(* Logix 5000 project; controller Sucrose_Main Emulate 5570 rev 20.12; software revision 20.01; part 20 of 30 *)
(* tags used below, declared in another part *)
   ClearFault_Master : BOOL;
   ClearFault_Master_TMR : TIMER;
   DATE_TIME : Date_Time;
   ONESHOTBITS : INT[10];
   Rung_Comment : BOOL;
   SucroseCIP_FILTRATION_REMOTE : CIP_REMOTE;
   SucroseDischarge : Area_Program;
   SucroseFiltration : Area_Program;
   TANK1_DATE_TIME : Date_Time;
   TANK2_DATE_TIME : Date_Time;
   TANK3_DATE_TIME : Date_Time;
   TK_23_01_01_RECEIVING_COMPLETE : BOOL;
   TK_23_02_01_RECEIVING_COMPLETE : BOOL;
   TK_23_03_01_RECEIVING_COMPLETE : BOOL;
(* Master_Main, continued *)

ROUTINE Date_Time   (* ladder *)
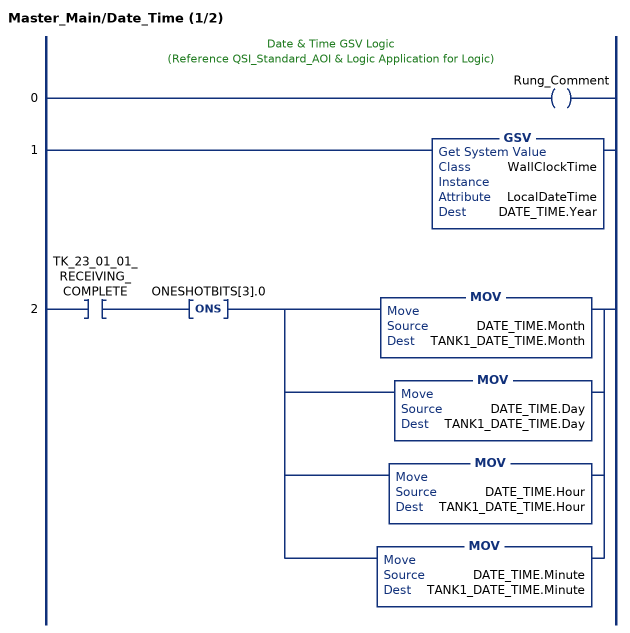
   // Date & Time GSV Logic
   // (Reference QSI_Standard_AOI & Logic Application for Logic)
   0: OTE(Rung_Comment);
   1: GSV(WallClockTime,,LocalDateTime,DATE_TIME.Year);
   2: XIC(TK_23_01_01_RECEIVING_COMPLETE)ONS(ONESHOTBITS[3].0)[MOV(DATE_TIME.Month,TANK1_DATE_TIME.Month) ,MOV(DATE_TIME.Day,TANK1_DATE_TIME.Day) ,MOV(DATE_TIME.Hour,TANK1_DATE_TIME.Hour) ,MOV(DATE_TIME.Minute,TANK1_DATE_TIME.Minute) ];
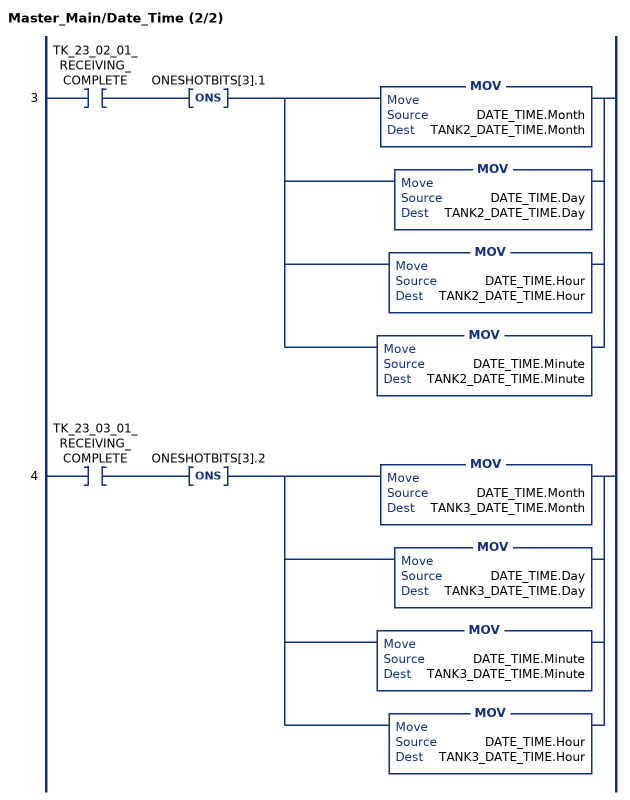
   3: XIC(TK_23_02_01_RECEIVING_COMPLETE)ONS(ONESHOTBITS[3].1)[MOV(DATE_TIME.Month,TANK2_DATE_TIME.Month) ,MOV(DATE_TIME.Day,TANK2_DATE_TIME.Day) ,MOV(DATE_TIME.Hour,TANK2_DATE_TIME.Hour) ,MOV(DATE_TIME.Minute,TANK2_DATE_TIME.Minute) ];
   4: XIC(TK_23_03_01_RECEIVING_COMPLETE)ONS(ONESHOTBITS[3].2)[MOV(DATE_TIME.Month,TANK3_DATE_TIME.Month) ,MOV(DATE_TIME.Day,TANK3_DATE_TIME.Day) ,MOV(DATE_TIME.Minute,TANK3_DATE_TIME.Minute) ,MOV(DATE_TIME.Hour,TANK3_DATE_TIME.Hour) ];
END_ROUTINE

ROUTINE Drive_ClearFault   (* ladder *)
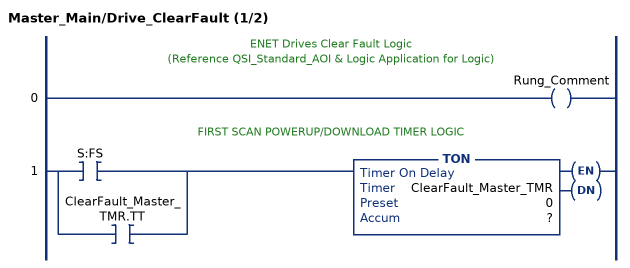
   // ENET Drives Clear Fault Logic
   // (Reference QSI_Standard_AOI & Logic Application for Logic)
   0: OTE(Rung_Comment);
   // FIRST SCAN POWERUP/DOWNLOAD TIMER LOGIC
   1: [XIC(S:FS) ,XIC(ClearFault_Master_TMR.TT) ]TON(ClearFault_Master_TMR,?,?);
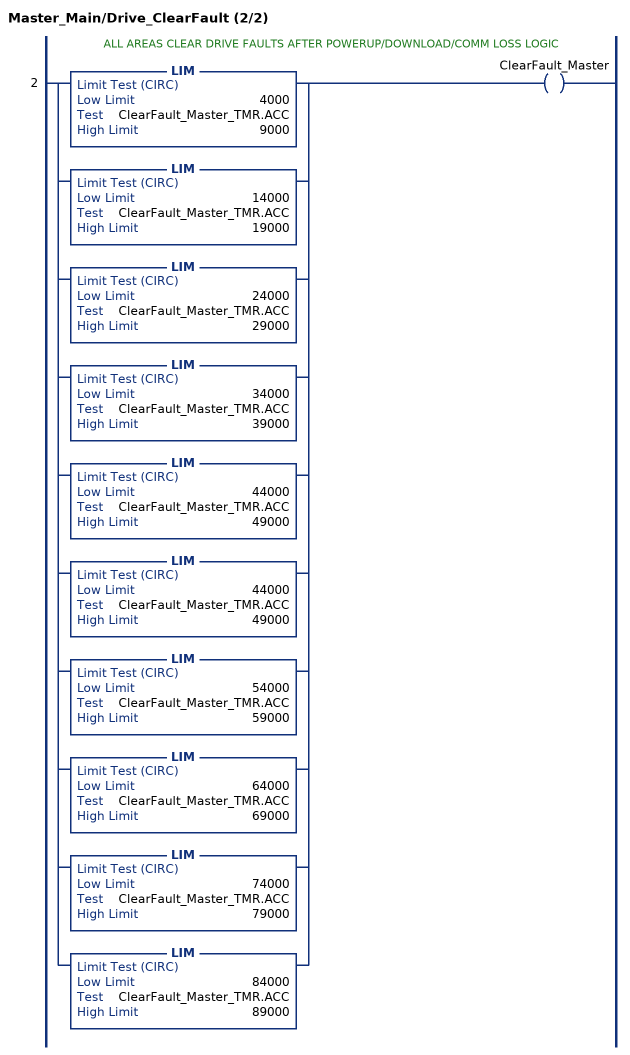
   // ALL AREAS CLEAR DRIVE FAULTS AFTER POWERUP/DOWNLOAD/COMM LOSS LOGIC
   2: [LIM(4000,ClearFault_Master_TMR.ACC,9000) ,LIM(14000,ClearFault_Master_TMR.ACC,19000) ,LIM(24000,ClearFault_Master_TMR.ACC,29000) ,LIM(34000,ClearFault_Master_TMR.ACC,39000) ,LIM(44000,ClearFault_Master_TMR.ACC,49000) ,LIM(44000,ClearFault_Master_TMR.ACC,49000) ,LIM(54000,ClearFault_Master_TMR.ACC,59000) ,LIM(64000,ClearFault_Master_TMR.ACC,69000) ,LIM(74000,ClearFault_Master_TMR.ACC,79000) ,LIM(84000,ClearFault_Master_TMR.ACC,89000) ]OTE(ClearFault_Master);
END_ROUTINE

ROUTINE HMI   (* ladder *)
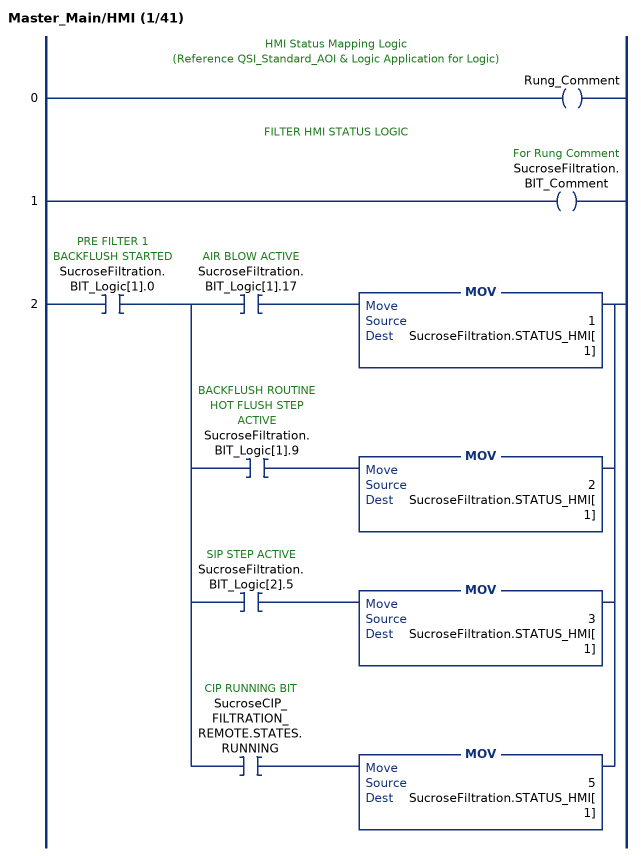
   // HMI Status Mapping Logic
   // (Reference QSI_Standard_AOI & Logic Application for Logic)
   0: OTE(Rung_Comment);
   // FILTER HMI STATUS LOGIC
   1: OTE(SucroseFiltration.BIT_Comment);
   2: XIC(SucroseFiltration.BIT_Logic[1].0)[XIC(SucroseFiltration.BIT_Logic[1].17) MOV(1,SucroseFiltration.STATUS_HMI[1]) ,XIC(SucroseFiltration.BIT_Logic[1].9) MOV(2,SucroseFiltration.STATUS_HMI[1]) ,XIC(SucroseFiltration.BIT_Logic[2].5) MOV(3,SucroseFiltration.STATUS_HMI[1]) ,XIC(SucroseCIP_FILTRATION_REMOTE.STATES.RUNNING) MOV(5,SucroseFiltration.STATUS_HMI[1]) ];
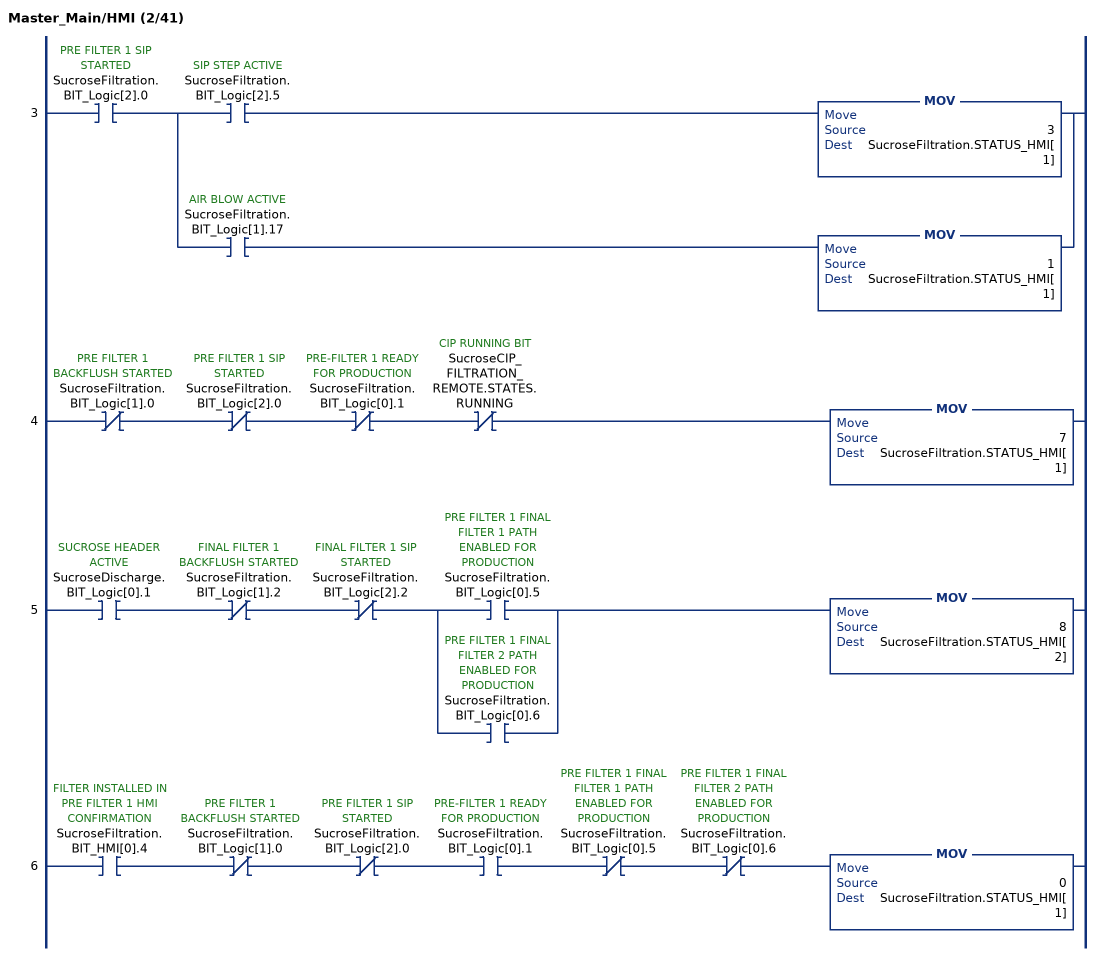
   3: XIC(SucroseFiltration.BIT_Logic[2].0)[XIC(SucroseFiltration.BIT_Logic[2].5) MOV(3,SucroseFiltration.STATUS_HMI[1]) ,XIC(SucroseFiltration.BIT_Logic[1].17) MOV(1,SucroseFiltration.STATUS_HMI[1]) ];
   4: XIO(SucroseFiltration.BIT_Logic[1].0)XIO(SucroseFiltration.BIT_Logic[2].0)XIO(SucroseFiltration.BIT_Logic[0].1)XIO(SucroseCIP_FILTRATION_REMOTE.STATES.RUNNING)MOV(7,SucroseFiltration.STATUS_HMI[1]);
   5: XIC(SucroseDischarge.BIT_Logic[0].1)XIO(SucroseFiltration.BIT_Logic[1].2)XIO(SucroseFiltration.BIT_Logic[2].2)[XIC(SucroseFiltration.BIT_Logic[0].5) ,XIC(SucroseFiltration.BIT_Logic[0].6) ]MOV(8,SucroseFiltration.STATUS_HMI[2]);
   6: XIC(SucroseFiltration.BIT_HMI[0].4)XIO(SucroseFiltration.BIT_Logic[1].0)XIO(SucroseFiltration.BIT_Logic[2].0)XIC(SucroseFiltration.BIT_Logic[0].1)XIO(SucroseFiltration.BIT_Logic[0].5)XIO(SucroseFiltration.BIT_Logic[0].6)MOV(0,SucroseFiltration.STATUS_HMI[1]);
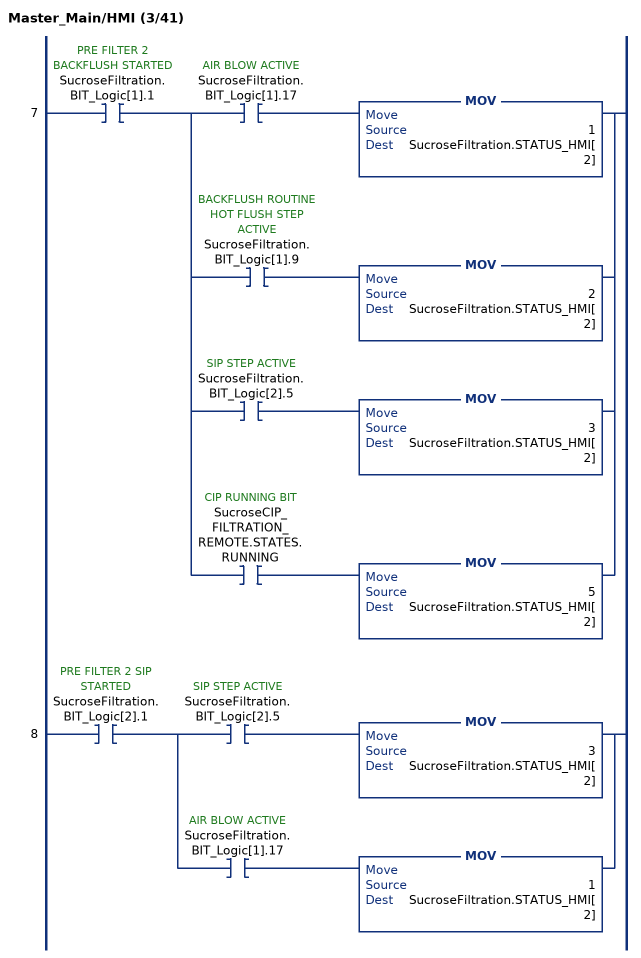
   7: XIC(SucroseFiltration.BIT_Logic[1].1)[XIC(SucroseFiltration.BIT_Logic[1].17) MOV(1,SucroseFiltration.STATUS_HMI[2]) ,XIC(SucroseFiltration.BIT_Logic[1].9) MOV(2,SucroseFiltration.STATUS_HMI[2]) ,XIC(SucroseFiltration.BIT_Logic[2].5) MOV(3,SucroseFiltration.STATUS_HMI[2]) ,XIC(SucroseCIP_FILTRATION_REMOTE.STATES.RUNNING) MOV(5,SucroseFiltration.STATUS_HMI[2]) ];
   8: XIC(SucroseFiltration.BIT_Logic[2].1)[XIC(SucroseFiltration.BIT_Logic[2].5) MOV(3,SucroseFiltration.STATUS_HMI[2]) ,XIC(SucroseFiltration.BIT_Logic[1].17) MOV(1,SucroseFiltration.STATUS_HMI[2]) ];
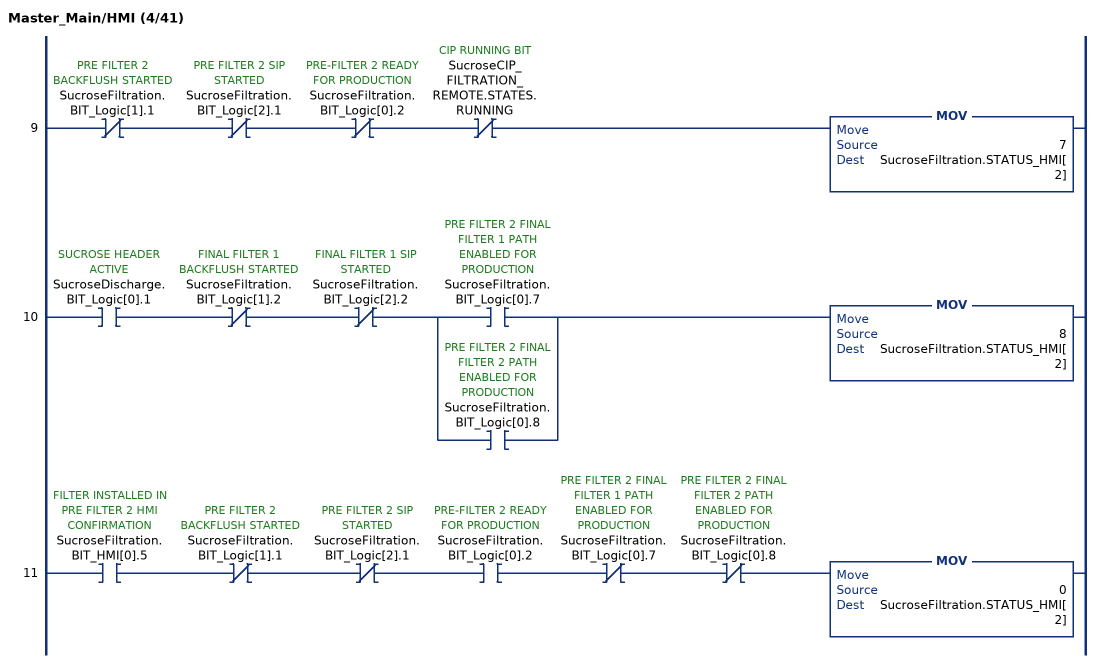
   9: XIO(SucroseFiltration.BIT_Logic[1].1)XIO(SucroseFiltration.BIT_Logic[2].1)XIO(SucroseFiltration.BIT_Logic[0].2)XIO(SucroseCIP_FILTRATION_REMOTE.STATES.RUNNING)MOV(7,SucroseFiltration.STATUS_HMI[2]);
   10: XIC(SucroseDischarge.BIT_Logic[0].1)XIO(SucroseFiltration.BIT_Logic[1].2)XIO(SucroseFiltration.BIT_Logic[2].2)[XIC(SucroseFiltration.BIT_Logic[0].7) ,XIC(SucroseFiltration.BIT_Logic[0].8) ]MOV(8,SucroseFiltration.STATUS_HMI[2]);
   11: XIC(SucroseFiltration.BIT_HMI[0].5)XIO(SucroseFiltration.BIT_Logic[1].1)XIO(SucroseFiltration.BIT_Logic[2].1)XIC(SucroseFiltration.BIT_Logic[0].2)XIO(SucroseFiltration.BIT_Logic[0].7)XIO(SucroseFiltration.BIT_Logic[0].8)MOV(0,SucroseFiltration.STATUS_HMI[2]);
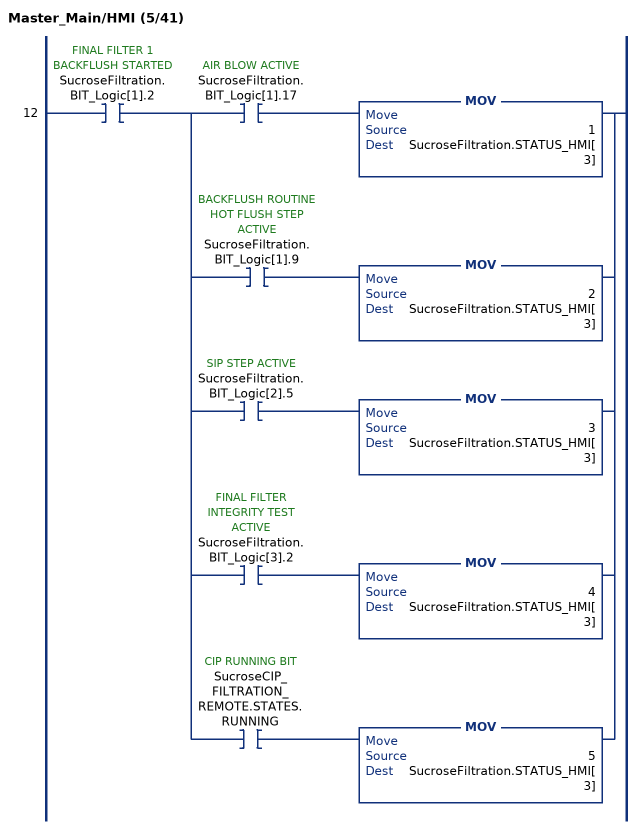
   12: XIC(SucroseFiltration.BIT_Logic[1].2)[XIC(SucroseFiltration.BIT_Logic[1].17) MOV(1,SucroseFiltration.STATUS_HMI[3]) ,XIC(SucroseFiltration.BIT_Logic[1].9) MOV(2,SucroseFiltration.STATUS_HMI[3]) ,XIC(SucroseFiltration.BIT_Logic[2].5) MOV(3,SucroseFiltration.STATUS_HMI[3]) ,XIC(SucroseFiltration.BIT_Logic[3].2) MOV(4,SucroseFiltration.STATUS_HMI[3]) ,XIC(SucroseCIP_FILTRATION_REMOTE.STATES.RUNNING) MOV(5,SucroseFiltration.STATUS_HMI[3]) ];
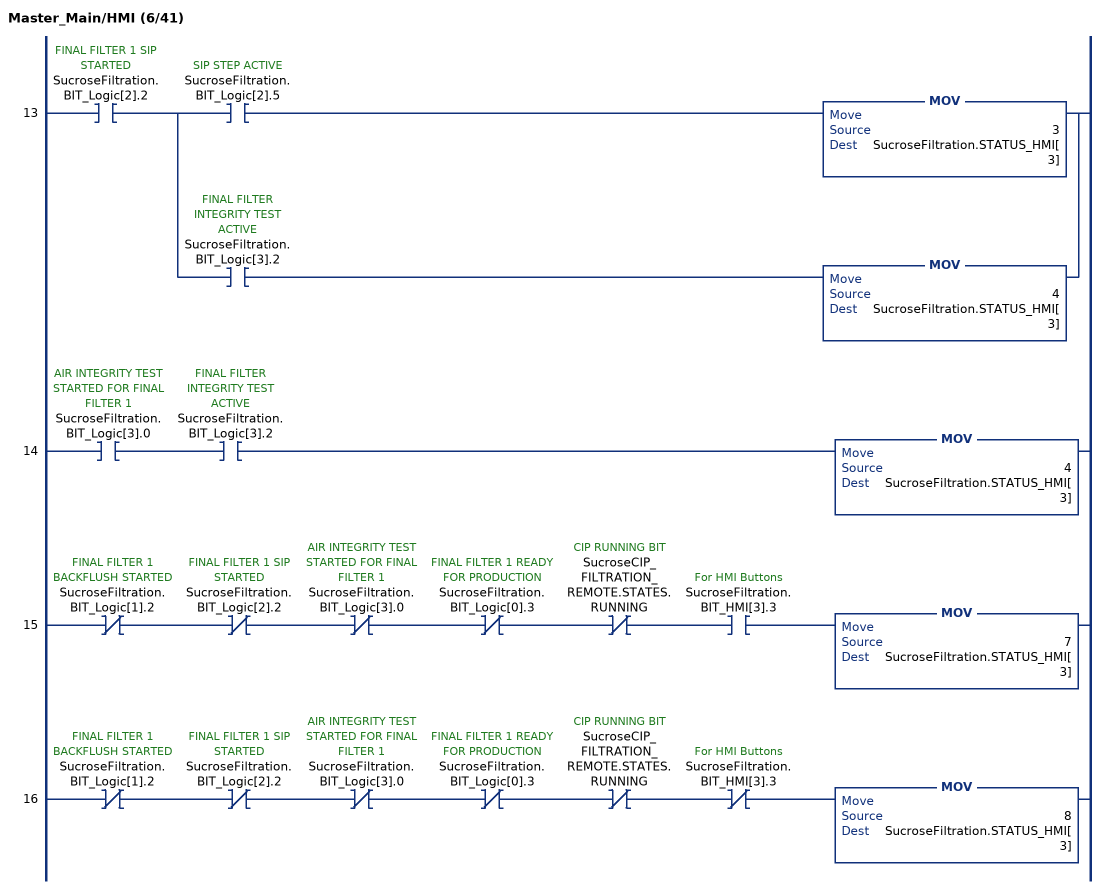
   13: XIC(SucroseFiltration.BIT_Logic[2].2)[XIC(SucroseFiltration.BIT_Logic[2].5) MOV(3,SucroseFiltration.STATUS_HMI[3]) ,XIC(SucroseFiltration.BIT_Logic[3].2) MOV(4,SucroseFiltration.STATUS_HMI[3]) ];
   14: XIC(SucroseFiltration.BIT_Logic[3].0)XIC(SucroseFiltration.BIT_Logic[3].2)MOV(4,SucroseFiltration.STATUS_HMI[3]);
   15: XIO(SucroseFiltration.BIT_Logic[1].2)XIO(SucroseFiltration.BIT_Logic[2].2)XIO(SucroseFiltration.BIT_Logic[3].0)XIO(SucroseFiltration.BIT_Logic[0].3)XIO(SucroseCIP_FILTRATION_REMOTE.STATES.RUNNING)XIC(SucroseFiltration.BIT_HMI[3].3)MOV(7,SucroseFiltration.STATUS_HMI[3]);
   16: XIO(SucroseFiltration.BIT_Logic[1].2)XIO(SucroseFiltration.BIT_Logic[2].2)XIO(SucroseFiltration.BIT_Logic[3].0)XIO(SucroseFiltration.BIT_Logic[0].3)XIO(SucroseCIP_FILTRATION_REMOTE.STATES.RUNNING)XIO(SucroseFiltration.BIT_HMI[3].3)MOV(8,SucroseFiltration.STATUS_HMI[3]);
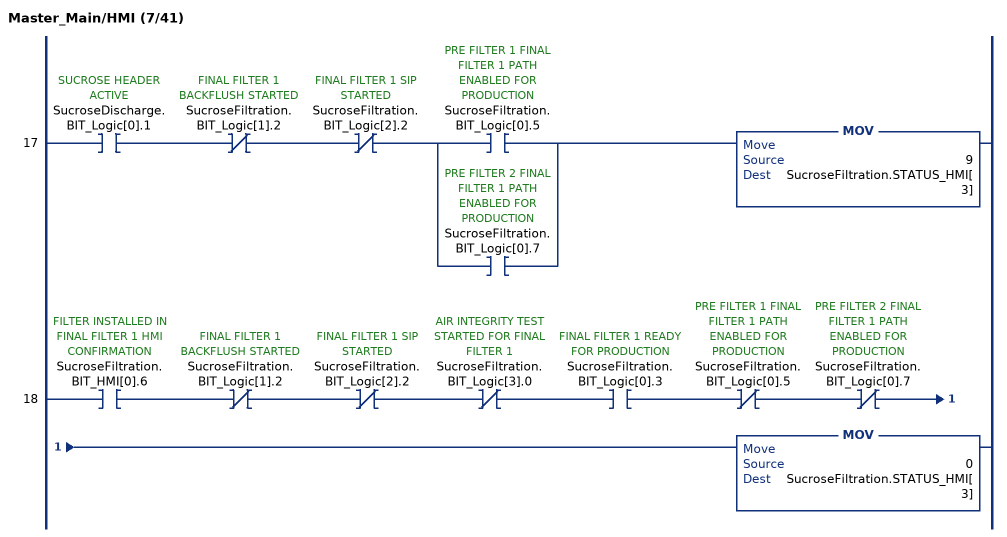
   17: XIC(SucroseDischarge.BIT_Logic[0].1)XIO(SucroseFiltration.BIT_Logic[1].2)XIO(SucroseFiltration.BIT_Logic[2].2)[XIC(SucroseFiltration.BIT_Logic[0].5) ,XIC(SucroseFiltration.BIT_Logic[0].7) ]MOV(9,SucroseFiltration.STATUS_HMI[3]);
   18: XIC(SucroseFiltration.BIT_HMI[0].6)XIO(SucroseFiltration.BIT_Logic[1].2)XIO(SucroseFiltration.BIT_Logic[2].2)XIO(SucroseFiltration.BIT_Logic[3].0)XIC(SucroseFiltration.BIT_Logic[0].3)XIO(SucroseFiltration.BIT_Logic[0].5)XIO(SucroseFiltration.BIT_Logic[0].7)MOV(0,SucroseFiltration.STATUS_HMI[3]);
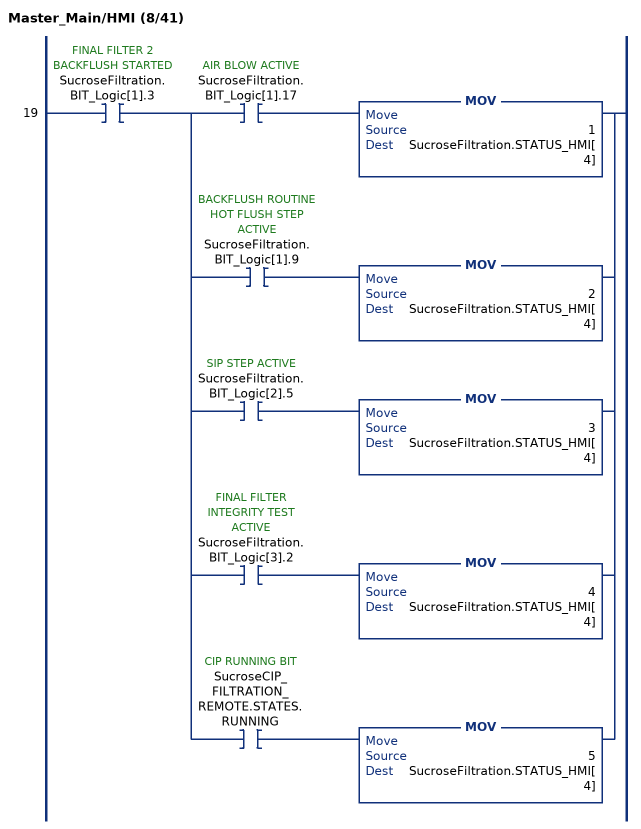
   19: XIC(SucroseFiltration.BIT_Logic[1].3)[XIC(SucroseFiltration.BIT_Logic[1].17) MOV(1,SucroseFiltration.STATUS_HMI[4]) ,XIC(SucroseFiltration.BIT_Logic[1].9) MOV(2,SucroseFiltration.STATUS_HMI[4]) ,XIC(SucroseFiltration.BIT_Logic[2].5) MOV(3,SucroseFiltration.STATUS_HMI[4]) ,XIC(SucroseFiltration.BIT_Logic[3].2) MOV(4,SucroseFiltration.STATUS_HMI[4]) ,XIC(SucroseCIP_FILTRATION_REMOTE.STATES.RUNNING) MOV(5,SucroseFiltration.STATUS_HMI[4]) ];
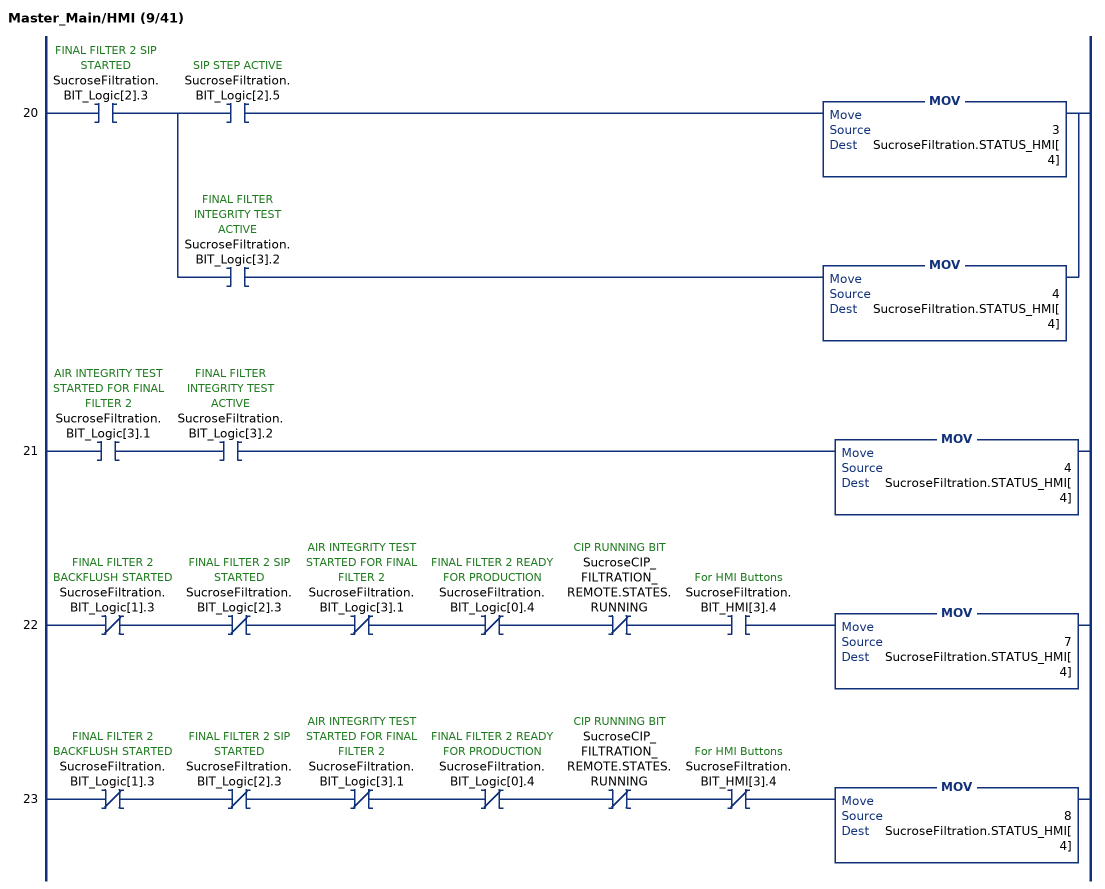
   20: XIC(SucroseFiltration.BIT_Logic[2].3)[XIC(SucroseFiltration.BIT_Logic[2].5) MOV(3,SucroseFiltration.STATUS_HMI[4]) ,XIC(SucroseFiltration.BIT_Logic[3].2) MOV(4,SucroseFiltration.STATUS_HMI[4]) ];
   21: XIC(SucroseFiltration.BIT_Logic[3].1)XIC(SucroseFiltration.BIT_Logic[3].2)MOV(4,SucroseFiltration.STATUS_HMI[4]);
   22: XIO(SucroseFiltration.BIT_Logic[1].3)XIO(SucroseFiltration.BIT_Logic[2].3)XIO(SucroseFiltration.BIT_Logic[3].1)XIO(SucroseFiltration.BIT_Logic[0].4)XIO(SucroseCIP_FILTRATION_REMOTE.STATES.RUNNING)XIC(SucroseFiltration.BIT_HMI[3].4)MOV(7,SucroseFiltration.STATUS_HMI[4]);
   23: XIO(SucroseFiltration.BIT_Logic[1].3)XIO(SucroseFiltration.BIT_Logic[2].3)XIO(SucroseFiltration.BIT_Logic[3].1)XIO(SucroseFiltration.BIT_Logic[0].4)XIO(SucroseCIP_FILTRATION_REMOTE.STATES.RUNNING)XIO(SucroseFiltration.BIT_HMI[3].4)MOV(8,SucroseFiltration.STATUS_HMI[4]);
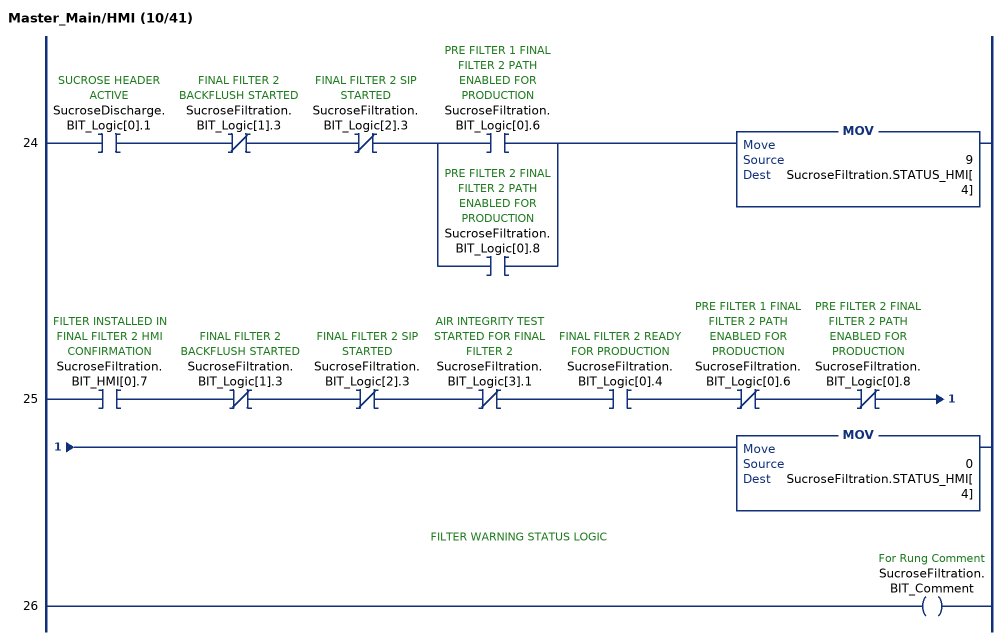
   24: XIC(SucroseDischarge.BIT_Logic[0].1)XIO(SucroseFiltration.BIT_Logic[1].3)XIO(SucroseFiltration.BIT_Logic[2].3)[XIC(SucroseFiltration.BIT_Logic[0].6) ,XIC(SucroseFiltration.BIT_Logic[0].8) ]MOV(9,SucroseFiltration.STATUS_HMI[4]);
   25: XIC(SucroseFiltration.BIT_HMI[0].7)XIO(SucroseFiltration.BIT_Logic[1].3)XIO(SucroseFiltration.BIT_Logic[2].3)XIO(SucroseFiltration.BIT_Logic[3].1)XIC(SucroseFiltration.BIT_Logic[0].4)XIO(SucroseFiltration.BIT_Logic[0].6)XIO(SucroseFiltration.BIT_Logic[0].8)MOV(0,SucroseFiltration.STATUS_HMI[4]);
   // FILTER WARNING STATUS LOGIC
   26: OTE(SucroseFiltration.BIT_Comment);
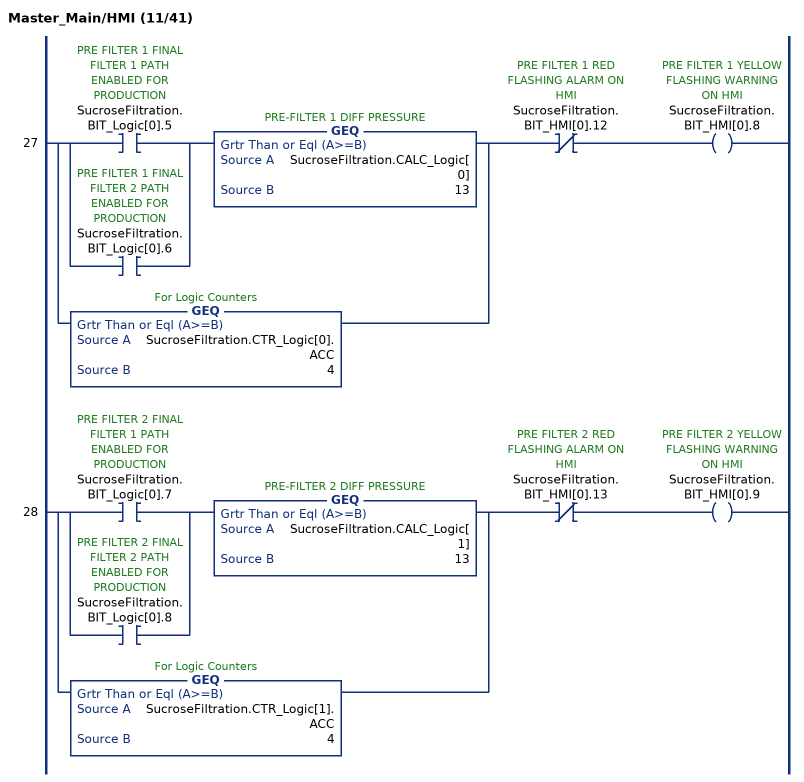
   27: [[XIC(SucroseFiltration.BIT_Logic[0].5) ,XIC(SucroseFiltration.BIT_Logic[0].6) ] GEQ(SucroseFiltration.CALC_Logic[0],13) ,GEQ(SucroseFiltration.CTR_Logic[0].ACC,4) ]XIO(SucroseFiltration.BIT_HMI[0].12)OTE(SucroseFiltration.BIT_HMI[0].8);
   28: [[XIC(SucroseFiltration.BIT_Logic[0].7) ,XIC(SucroseFiltration.BIT_Logic[0].8) ] GEQ(SucroseFiltration.CALC_Logic[1],13) ,GEQ(SucroseFiltration.CTR_Logic[1].ACC,4) ]XIO(SucroseFiltration.BIT_HMI[0].13)OTE(SucroseFiltration.BIT_HMI[0].9);
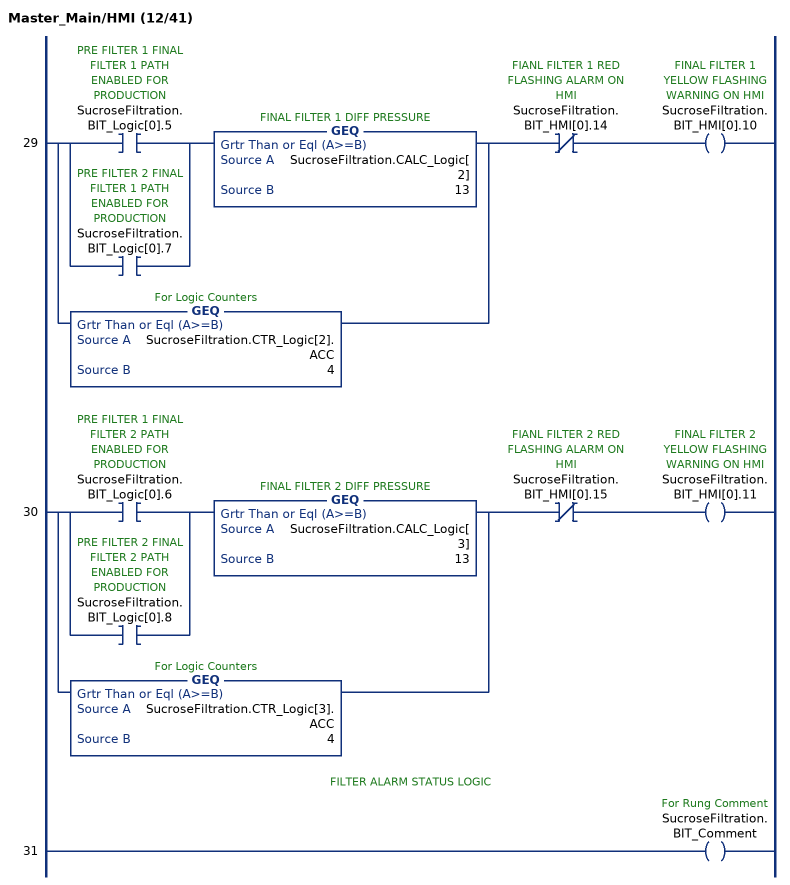
   29: [[XIC(SucroseFiltration.BIT_Logic[0].5) ,XIC(SucroseFiltration.BIT_Logic[0].7) ] GEQ(SucroseFiltration.CALC_Logic[2],13) ,GEQ(SucroseFiltration.CTR_Logic[2].ACC,4) ]XIO(SucroseFiltration.BIT_HMI[0].14)OTE(SucroseFiltration.BIT_HMI[0].10);
   30: [[XIC(SucroseFiltration.BIT_Logic[0].6) ,XIC(SucroseFiltration.BIT_Logic[0].8) ] GEQ(SucroseFiltration.CALC_Logic[3],13) ,GEQ(SucroseFiltration.CTR_Logic[3].ACC,4) ]XIO(SucroseFiltration.BIT_HMI[0].15)OTE(SucroseFiltration.BIT_HMI[0].11);
   // FILTER ALARM STATUS LOGIC
   31: OTE(SucroseFiltration.BIT_Comment);
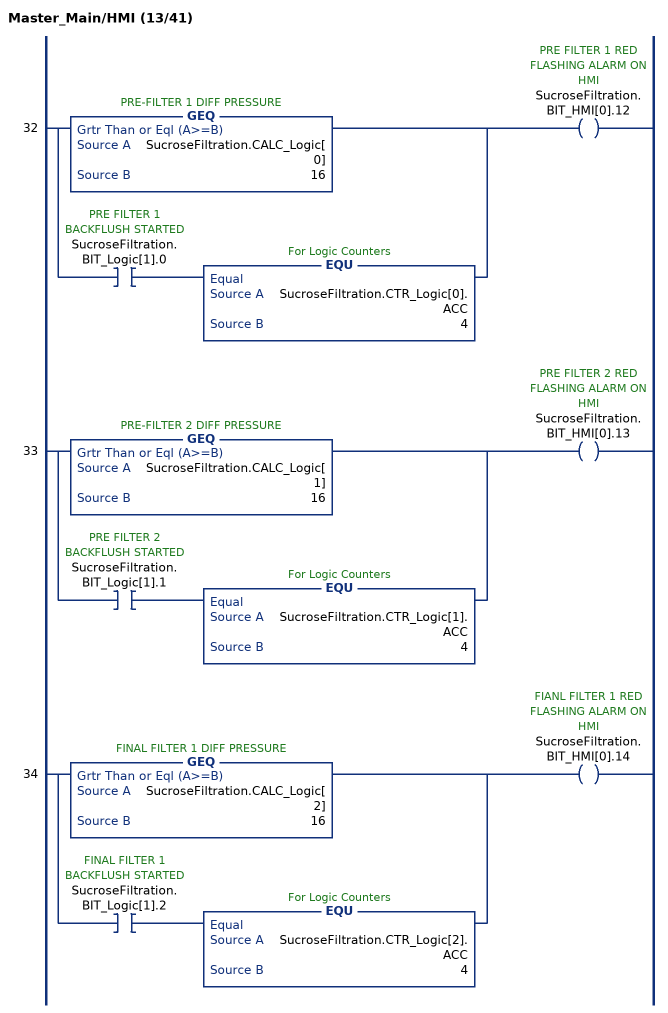
   32: [GEQ(SucroseFiltration.CALC_Logic[0],16) ,XIC(SucroseFiltration.BIT_Logic[1].0) EQU(SucroseFiltration.CTR_Logic[0].ACC,4) ]OTE(SucroseFiltration.BIT_HMI[0].12);
   33: [GEQ(SucroseFiltration.CALC_Logic[1],16) ,XIC(SucroseFiltration.BIT_Logic[1].1) EQU(SucroseFiltration.CTR_Logic[1].ACC,4) ]OTE(SucroseFiltration.BIT_HMI[0].13);
   34: [GEQ(SucroseFiltration.CALC_Logic[2],16) ,XIC(SucroseFiltration.BIT_Logic[1].2) EQU(SucroseFiltration.CTR_Logic[2].ACC,4) ]OTE(SucroseFiltration.BIT_HMI[0].14);
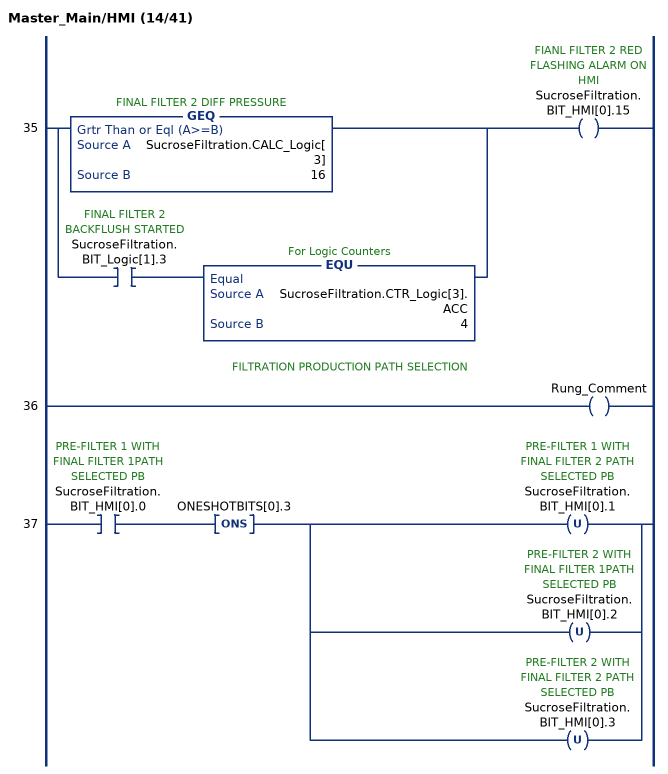
   35: [GEQ(SucroseFiltration.CALC_Logic[3],16) ,XIC(SucroseFiltration.BIT_Logic[1].3) EQU(SucroseFiltration.CTR_Logic[3].ACC,4) ]OTE(SucroseFiltration.BIT_HMI[0].15);
   // FILTRATION PRODUCTION PATH SELECTION
   36: OTE(Rung_Comment);
   37: XIC(SucroseFiltration.BIT_HMI[0].0)ONS(ONESHOTBITS[0].3)[OTU(SucroseFiltration.BIT_HMI[0].1) ,OTU(SucroseFiltration.BIT_HMI[0].2) ,OTU(SucroseFiltration.BIT_HMI[0].3) ];
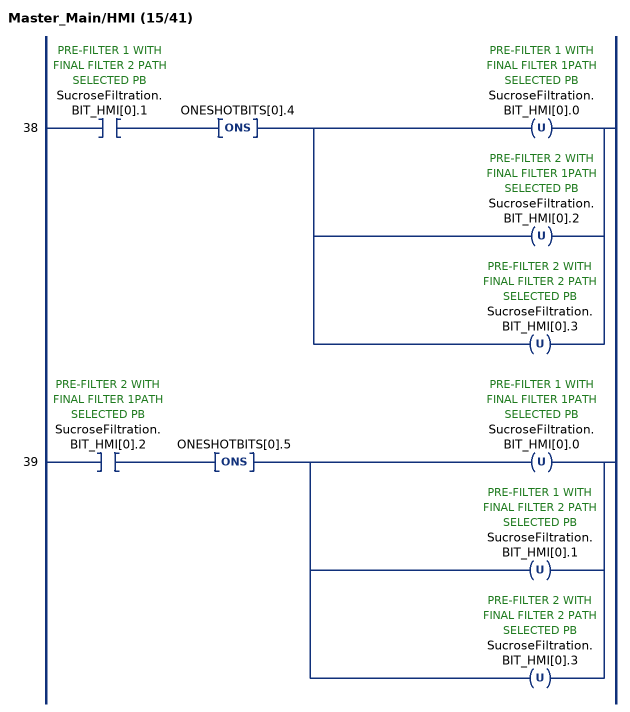
   38: XIC(SucroseFiltration.BIT_HMI[0].1)ONS(ONESHOTBITS[0].4)[OTU(SucroseFiltration.BIT_HMI[0].0) ,OTU(SucroseFiltration.BIT_HMI[0].2) ,OTU(SucroseFiltration.BIT_HMI[0].3) ];
   39: XIC(SucroseFiltration.BIT_HMI[0].2)ONS(ONESHOTBITS[0].5)[OTU(SucroseFiltration.BIT_HMI[0].0) ,OTU(SucroseFiltration.BIT_HMI[0].1) ,OTU(SucroseFiltration.BIT_HMI[0].3) ];
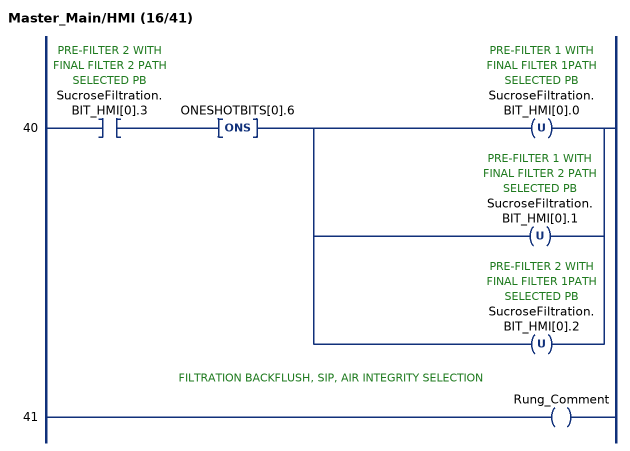
   40: XIC(SucroseFiltration.BIT_HMI[0].3)ONS(ONESHOTBITS[0].6)[OTU(SucroseFiltration.BIT_HMI[0].0) ,OTU(SucroseFiltration.BIT_HMI[0].1) ,OTU(SucroseFiltration.BIT_HMI[0].2) ];
   // FILTRATION BACKFLUSH, SIP, AIR INTEGRITY SELECTION
   41: OTE(Rung_Comment);
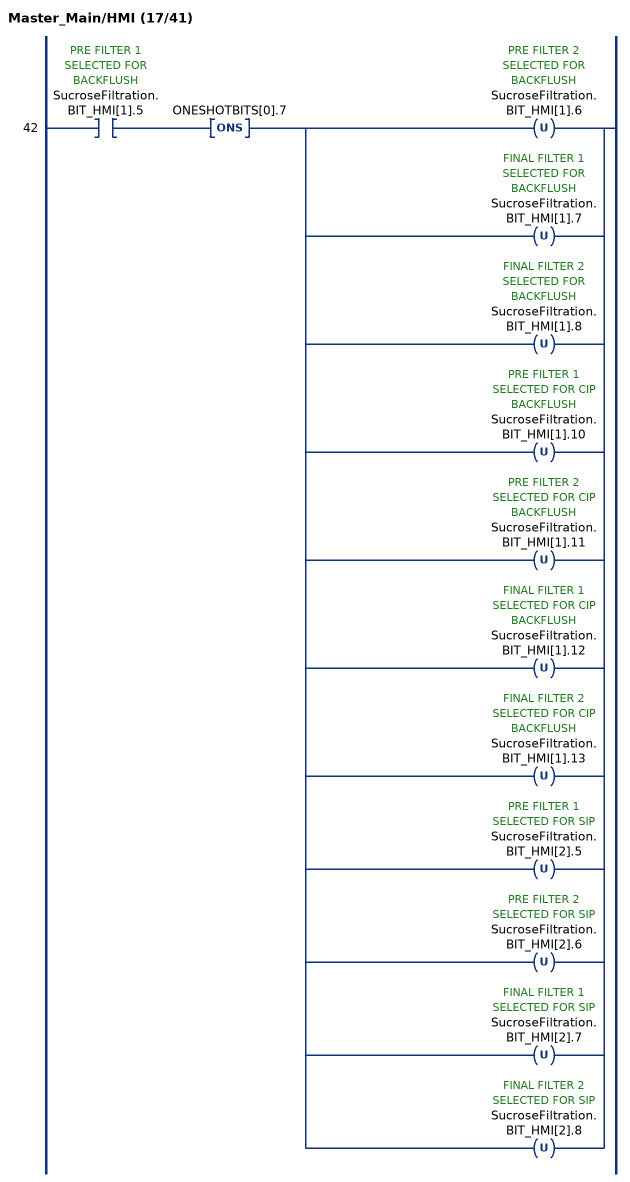
   42: XIC(SucroseFiltration.BIT_HMI[1].5)ONS(ONESHOTBITS[0].7)[OTU(SucroseFiltration.BIT_HMI[1].6) ,OTU(SucroseFiltration.BIT_HMI[1].7) ,OTU(SucroseFiltration.BIT_HMI[1].8) ,OTU(SucroseFiltration.BIT_HMI[1].10) ,OTU(SucroseFiltration.BIT_HMI[1].11) ,OTU(SucroseFiltration.BIT_HMI[1].12) ,OTU(SucroseFiltration.BIT_HMI[1].13) ,OTU(SucroseFiltration.BIT_HMI[2].5) ,OTU(SucroseFiltration.BIT_HMI[2].6) ,OTU(SucroseFiltration.BIT_HMI[2].7) ,OTU(SucroseFiltration.BIT_HMI[2].8) ];
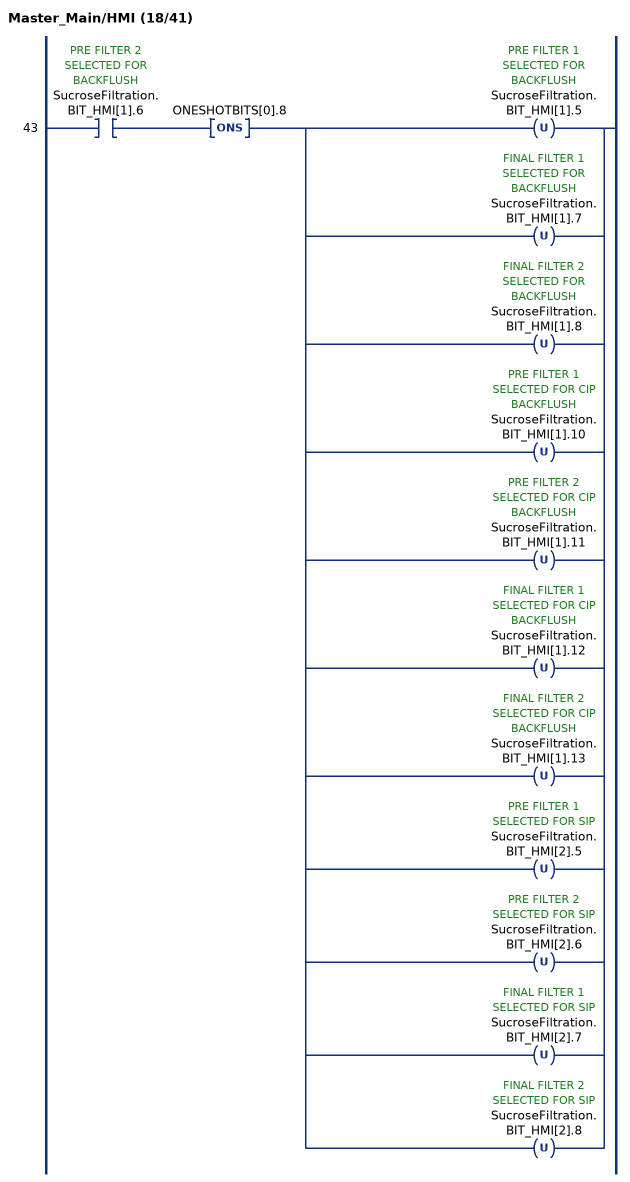
   43: XIC(SucroseFiltration.BIT_HMI[1].6)ONS(ONESHOTBITS[0].8)[OTU(SucroseFiltration.BIT_HMI[1].5) ,OTU(SucroseFiltration.BIT_HMI[1].7) ,OTU(SucroseFiltration.BIT_HMI[1].8) ,OTU(SucroseFiltration.BIT_HMI[1].10) ,OTU(SucroseFiltration.BIT_HMI[1].11) ,OTU(SucroseFiltration.BIT_HMI[1].12) ,OTU(SucroseFiltration.BIT_HMI[1].13) ,OTU(SucroseFiltration.BIT_HMI[2].5) ,OTU(SucroseFiltration.BIT_HMI[2].6) ,OTU(SucroseFiltration.BIT_HMI[2].7) ,OTU(SucroseFiltration.BIT_HMI[2].8) ];
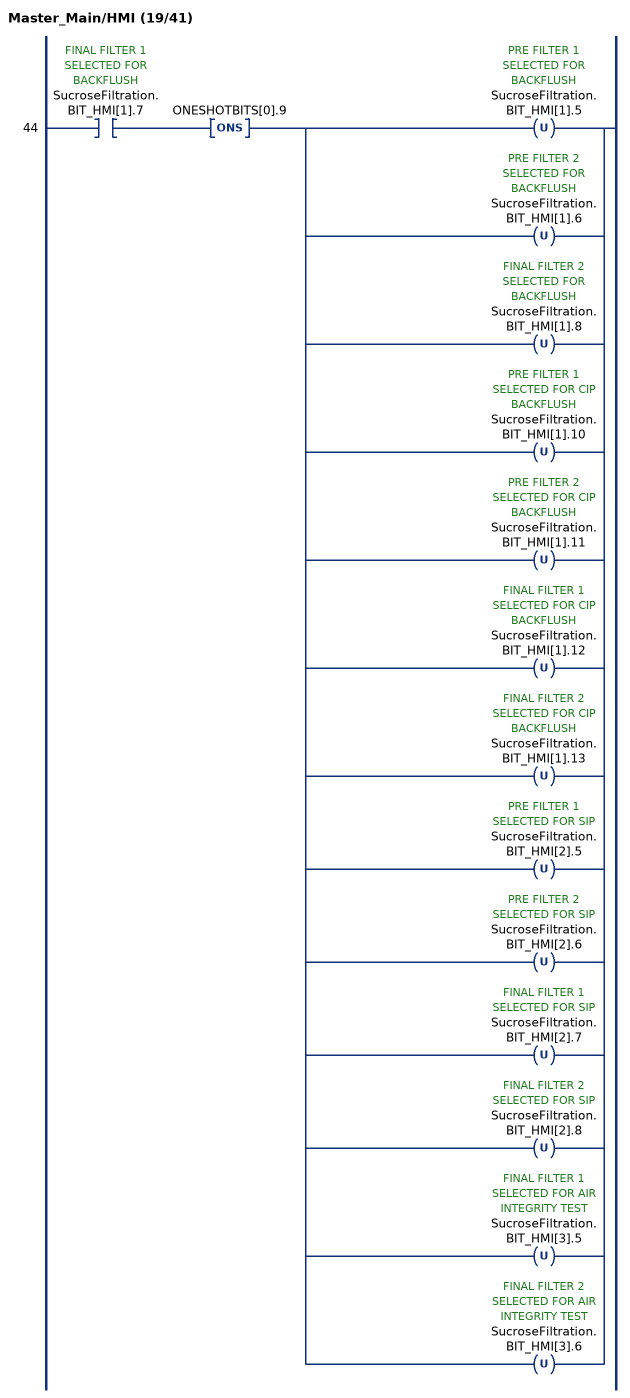
   44: XIC(SucroseFiltration.BIT_HMI[1].7)ONS(ONESHOTBITS[0].9)[OTU(SucroseFiltration.BIT_HMI[1].5) ,OTU(SucroseFiltration.BIT_HMI[1].6) ,OTU(SucroseFiltration.BIT_HMI[1].8) ,OTU(SucroseFiltration.BIT_HMI[1].10) ,OTU(SucroseFiltration.BIT_HMI[1].11) ,OTU(SucroseFiltration.BIT_HMI[1].12) ,OTU(SucroseFiltration.BIT_HMI[1].13) ,OTU(SucroseFiltration.BIT_HMI[2].5) ,OTU(SucroseFiltration.BIT_HMI[2].6) ,OTU(SucroseFiltration.BIT_HMI[2].7) ,OTU(SucroseFiltration.BIT_HMI[2].8) ,OTU(SucroseFiltration.BIT_HMI[3].5) ,OTU(SucroseFiltration.BIT_HMI[3].6) ];
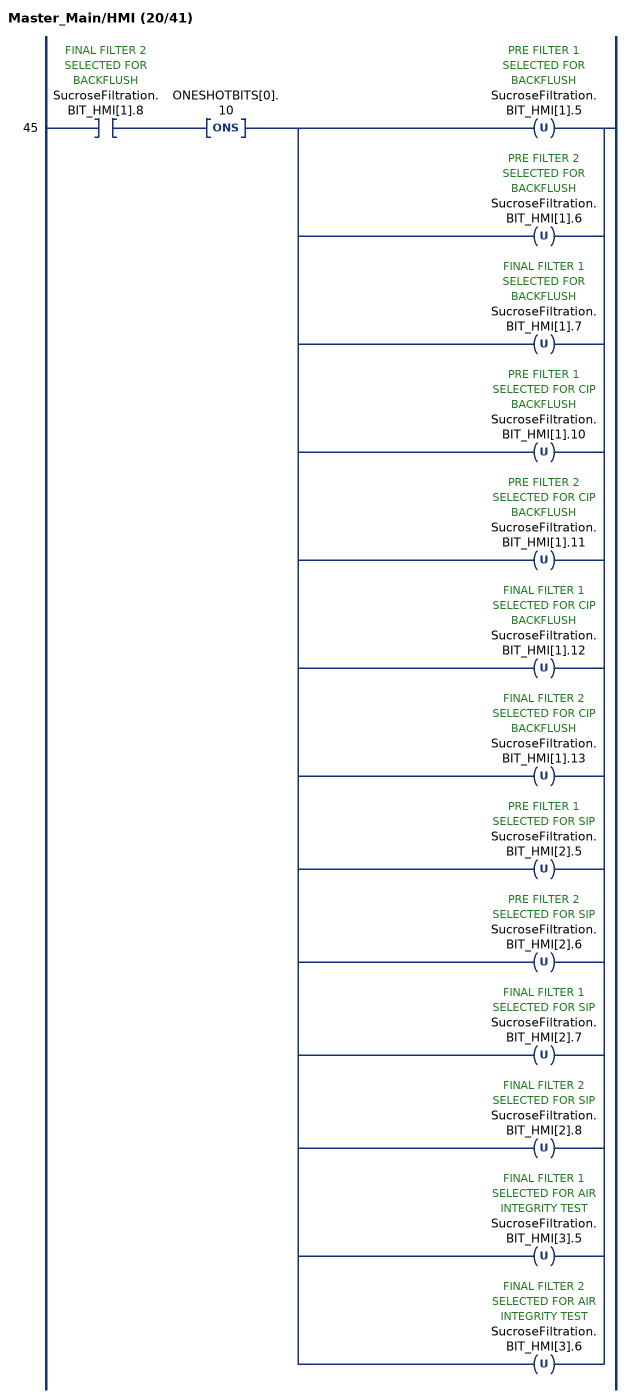
   45: XIC(SucroseFiltration.BIT_HMI[1].8)ONS(ONESHOTBITS[0].10)[OTU(SucroseFiltration.BIT_HMI[1].5) ,OTU(SucroseFiltration.BIT_HMI[1].6) ,OTU(SucroseFiltration.BIT_HMI[1].7) ,OTU(SucroseFiltration.BIT_HMI[1].10) ,OTU(SucroseFiltration.BIT_HMI[1].11) ,OTU(SucroseFiltration.BIT_HMI[1].12) ,OTU(SucroseFiltration.BIT_HMI[1].13) ,OTU(SucroseFiltration.BIT_HMI[2].5) ,OTU(SucroseFiltration.BIT_HMI[2].6) ,OTU(SucroseFiltration.BIT_HMI[2].7) ,OTU(SucroseFiltration.BIT_HMI[2].8) ,OTU(SucroseFiltration.BIT_HMI[3].5) ,OTU(SucroseFiltration.BIT_HMI[3].6) ];
